(* Logix 5000 project; controller Modbus_TCP_Client_Example vendor 1 type 14 code 154 rev 32.15; software revision 32.05; part 6 of 10 *)

ADD_ON_INSTRUCTION AMP_Point_to_Point_IO_Servo   (* revision 1.0, vendor Applied Motion Products Inc. *)
// Applied Motion - Point to Point Move with IO AOI
// Help:
// The Point-to-Point Move with I/O AOI executes moves involving up to 2 Input conditions and a possible output state change. The move variant can be any of the following:
// - FS - Feed to Sensor
// - FD - Feed to Double Sensor
// - FM - Feed to Sensor with Mask Distance
// - FY - Feed to Sensor with Safety Distance
// - FO - Feed to Length and Set Output
// - SH - Seek Home
// All six(6) of the above variants need exactly one I/O point except for FD which requires a second I/O point to be specified in the parameters.
VAR_IN_OUT
   Input : DINT[20]; {required}   // Drive Input Assembly
        [16]   // Analog_Input1
        [4]   // Alarm_Code
        [0]   // Control_Word_Received
        [10]   // Position_Error
        [11]   // Actual_Velocity_RPS
        [12]   // Digital_Outputs
        [13]   // Digital_Inputs
        [14]   // Analog_Output1
        [15]   // Analog_Output2
        [17]   // Analog_Input2
        [18]   // Torque_Limit
        [19]   // Second_Encoder_Speed
        [1]   // OpCode1_Received
        [2]   // Control_Mode
        [3]   // Status_Code
        [5]   // Supply_Voltage
        [6]   // Applied_Torque
        [7]   // Drive_Temperature
        [8]   // Encoder_Position
        [9]   // Second_Encoder_Position
   Output : DINT[11]; {required}   // Drive Output Assembly
        [10]   // Reserved
        [4]   // Target Velocity
        [0]   // Control Word
        [3]   // Target Pos
        [1]   // OpCode 1
        [2]   // OpCode 2
        [5]   // Porifle Acceleration
        [6]   // Profile Deceleration
        [7]   // Target Torque
        [8]   // OpCode 3
        [9]   // OpCode 4
END_VAR
VAR_INPUT
   Start : BOOL; {required}   // Start the Move
   Command : INT := 'FS'; {required}   // Command variant: FS/FD/FY/FM/FO/SH
   IO1_Number : DINT; {required}   // Main Input/Output Number (0 = Encoder index, 1-8 = In/Out 1-8)
   IO1_Condition : SINT := 'R'; {required}   // Main Input/Output Condition/State H/L/R/F (High/Low/Rising Edge/Falling Edge)
   IO2_Number : DINT; {required}   // Second Input/Output Number (0 = Encoder index, 1-8 = In/Out 1-8)
   IO2_Condition : SINT; {required}   // Second Input/Output Condition/State H/L/R/F (High/Low/Rising Edge/Falling Edge)
   Distance : DINT; {required}   // Distance to Move (negative = reverse)
   Speed : REAL; {required}   // Velocity of Move (rev/sec)
   Acc : REAL; {required}   // Acceleration of Move (rev/s/s)
   Dec : REAL; {required}   // Deceleration (rev/s/s)
   Change_Distance : DINT; {required}   // Change Distance (steps, FY/FM/FO only)
   Change_Speed : REAL; {required}   // Velocity Change (rev/s) (FD only)
END_VAR
VAR_OUTPUT
   Sent : BOOL; {access Read Only, visible}   // Move has been sent to drive
   In_Progress : BOOL; {access Read Only, visible}   // Move in progress
   Done : BOOL; {access Read Only, visible}   // Move completed without errors - desired position reached
   Error : BOOL; {access Read Only, visible}   // Move failed to complete - drive not ready or faulted
   State : DINT := 10; {access Read Only}   // Internal state of progress
END_VAR
VAR
   Loc_StatusCode : AMP_Status_Word_Servo; {access None}
   Loc_Start_ONS : BOOL; {access None}
   Loc_Input_Assembly : AMP_Input_Assembly_Servo_v2; {access None}
   Loc_Command_Timeout : TIMER := (PRE := 2000); {access None}   // Timer to output fault if command is not Done
   Loc_ChangeSpeed_Required : BOOL; {access None}
   Loc_ChangeDistance_Required : BOOL; {access None}
   Loc_IO2_Number_Encoded : DINT; {access None}
   Loc_IO2_Condition_Encoded : DINT; {access None}
   Loc_IO1_Condition_Encoded : DINT; {access None}
   Loc_IO1_Number_Encoded : DINT; {access None}
END_VAR

ROUTINE Logic   (* ladder *)
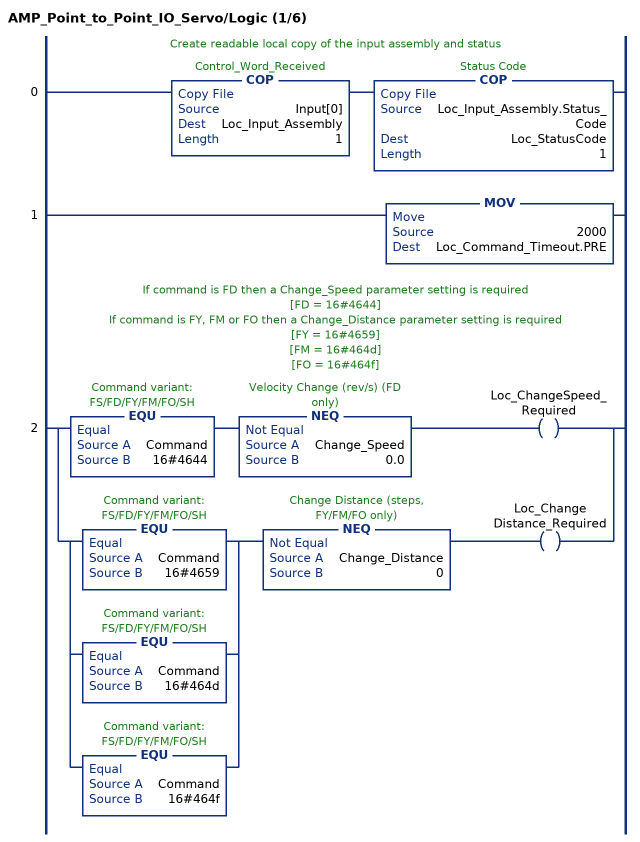
   // Create readable local copy of the input assembly and status
   0: COP(Input[0],Loc_Input_Assembly,1)COP(Loc_Input_Assembly.Status_Code,Loc_StatusCode,1);
   1: MOV(2000,Loc_Command_Timeout.PRE);
   // If command is FD then a Change_Speed parameter setting is required
   // [FD = 16#4644]
   // If command is FY, FM or FO then a Change_Distance parameter setting is required
   // [FY = 16#4659]
   // [FM = 16#464d]
   // [FO = 16#464f]
   2: [EQU(Command,16#4644) NEQ(Change_Speed,0.0) OTE(Loc_ChangeSpeed_Required) ,[EQU(Command,16#4659) ,EQU(Command,16#464d) ,EQU(Command,16#464f) ] NEQ(Change_Distance,0) OTE(Loc_ChangeDistance_Required) ];
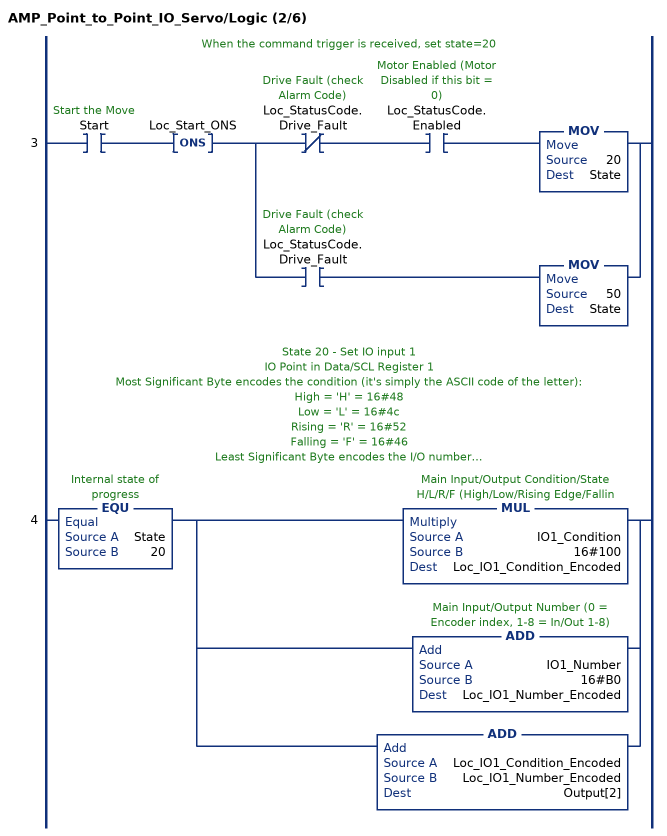
   // When the command trigger is received, set state=20
   3: XIC(Start)ONS(Loc_Start_ONS)[XIO(Loc_StatusCode.Drive_Fault) XIC(Loc_StatusCode.Enabled) MOV(20,State) ,XIC(Loc_StatusCode.Drive_Fault) MOV(50,State) ];
   // State 20 - Set IO input 1
   // IO Point in Data/SCL Register 1
   // Most Significant Byte encodes the condition (it's simply the ASCII code of the letter):
   // High = 'H' = 16#48
   // Low = 'L' = 16#4c
   // Rising = 'R' = 16#52
   // Falling = 'F' = 16#46
   // Least Significant Byte encodes the I/O number:
   // 0xB0-0xBC for connector  (IN/OUT1) depending on provided I/O number 0-12 (0=encoder)
   4: EQU(State,20)[MUL(IO1_Condition,16#100,Loc_IO1_Condition_Encoded) ,ADD(IO1_Number,16#B0,Loc_IO1_Number_Encoded) ,ADD(Loc_IO1_Condition_Encoded,Loc_IO1_Number_Encoded,Output[2]) ];
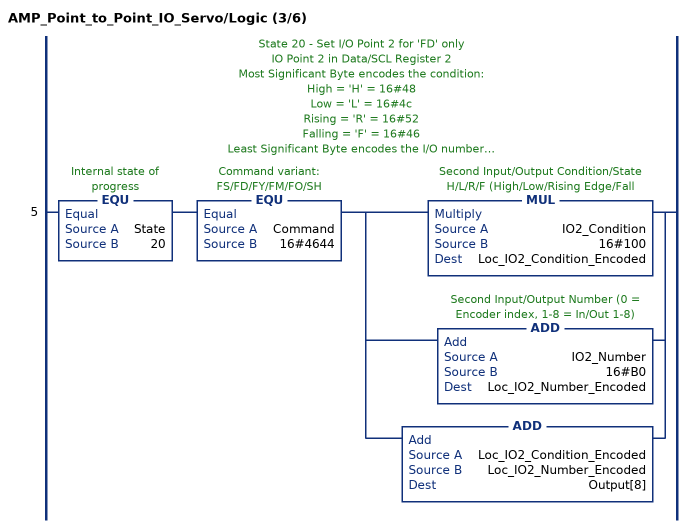
   // State 20 - Set I/O Point 2 for 'FD' only
   // IO Point 2 in Data/SCL Register 2
   // Most Significant Byte encodes the condition:
   // High = 'H' = 16#48
   // Low = 'L' = 16#4c
   // Rising = 'R' = 16#52
   // Falling = 'F' = 16#46
   // Least Significant Byte encodes the I/O number:
   // 0xB0-0xBC for connector  (IN/OUT1) depending on provided I/O number 0-12 (0=encoder)
   5: EQU(State,20)EQU(Command,16#4644)[MUL(IO2_Condition,16#100,Loc_IO2_Condition_Encoded) ,ADD(IO2_Number,16#B0,Loc_IO2_Number_Encoded) ,ADD(Loc_IO2_Condition_Encoded,Loc_IO2_Number_Encoded,Output[8]) ];
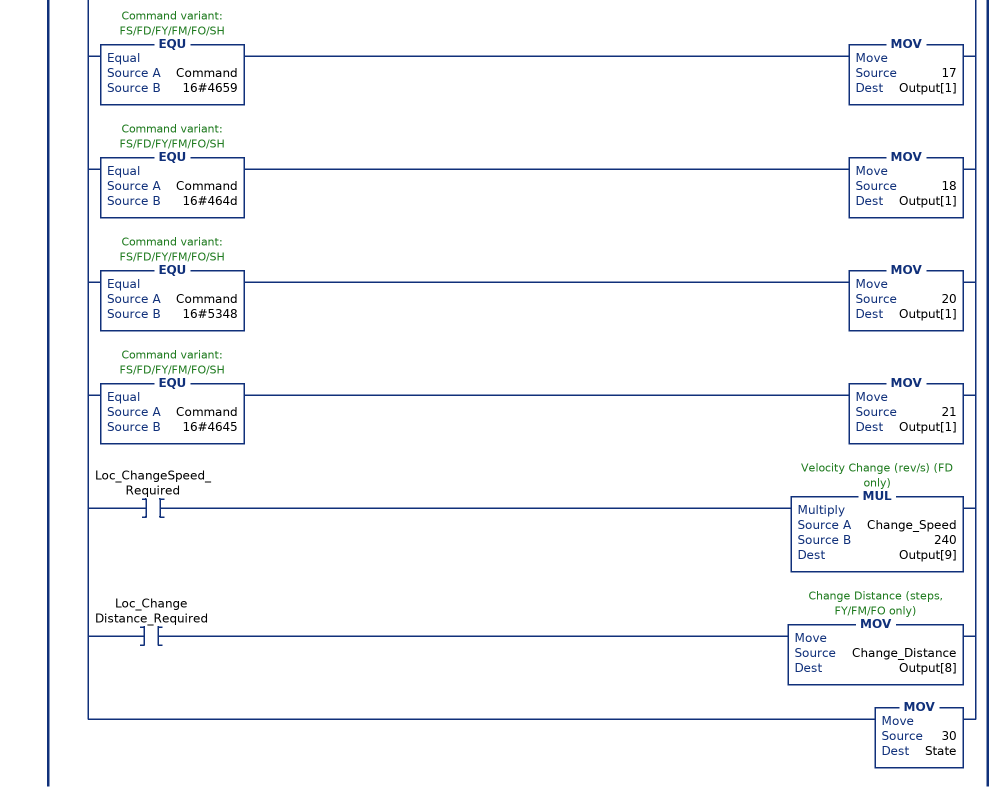
   // State 20 -
   // Distance in motor steps, no conversion required
   // Speed in rev/s, converted to 0.25 rev/min
   // Acceleration in rev/s/s, converted to 10 rev/min/s
   // Deceleration in rev/s/s, converted to 10 rev/min/s
   // FS (Feed to Sensor): ASCII = 16#4653, Cmd = 12,
   // FO (Feed to Length and Set Output): ASCII = 16#464f, Cmd = 13,
   // FD (Feed to Double Sensor): ASCII = 16#4644, Cmd = 16,
   // FY (Feed to Sensor with Safety Distance): ASCII = 16#4659, Cmd = 17,
   // FM (Feed to Sensor with Mask Distance): ASCII = 16#464d, Cmd = 18,
   // SH (Seek Home): ASCII = 16#5348, Cmd = 20
   6: EQU(State,20)EQU(Loc_Input_Assembly.Control_Mode,21)ADD(Loc_Input_Assembly.Control_Word_Received,1,Output[0])[MOV(Distance,Output[3]) ,MUL(Speed,240,Output[4]) ,MUL(Acc,6,Output[5]) ,MUL(Dec,6,Output[6]) ][[EQU(Command,16#4653) MOV(12,Output[1]) ,EQU(Command,16#464f) MOV(13,Output[1]) ,EQU(Command,16#4644) MOV(16,Output[1]) ,EQU(Command,16#4659) MOV(17,Output[1]) ,EQU(Command,16#464d) MOV(18,Output[1]) ,EQU(Command,16#5348) MOV(20,Output[1]) ,EQU(Command,16#4645) MOV(21,Output[1]) ] ,XIC(Loc_ChangeSpeed_Required) MUL(Change_Speed,240,Output[9]) ,XIC(Loc_ChangeDistance_Required) MOV(Change_Distance,Output[8]) ,MOV(30,State) ];
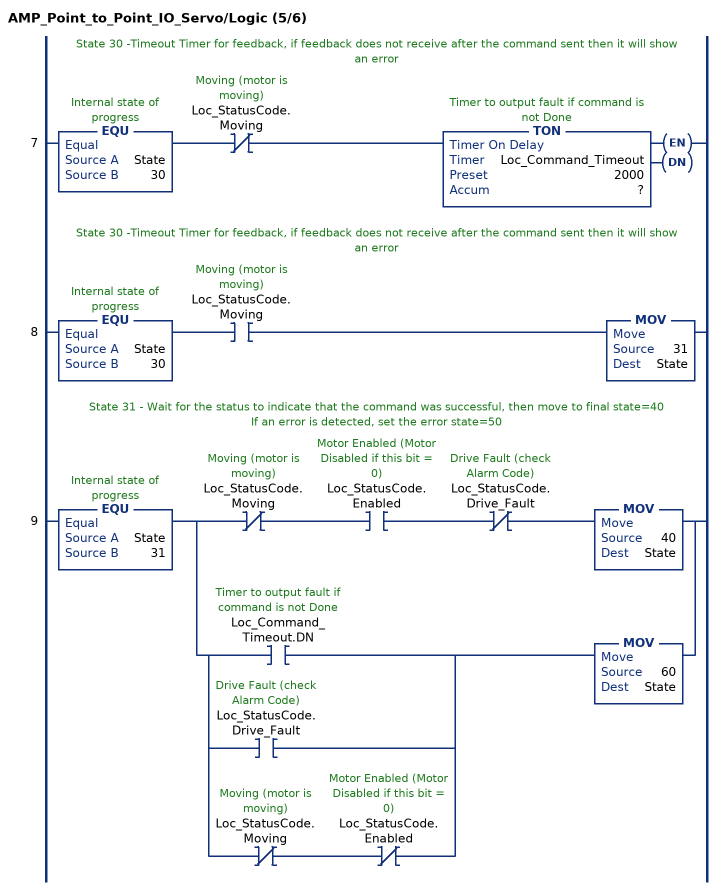
   // State 30 -Timeout Timer for feedback, if feedback does not receive after the command sent then it will show an error
   7: EQU(State,30)XIO(Loc_StatusCode.Moving)TON(Loc_Command_Timeout,?,?);
   // State 30 -Timeout Timer for feedback, if feedback does not receive after the command sent then it will show an error
   8: EQU(State,30)XIC(Loc_StatusCode.Moving)MOV(31,State);
   // State 31 - Wait for the status to indicate that the command was successful, then move to final state=40
   // If an error is detected, set the error state=50
   9: EQU(State,31)[XIO(Loc_StatusCode.Moving) XIC(Loc_StatusCode.Enabled) XIO(Loc_StatusCode.Drive_Fault) MOV(40,State) ,[XIC(Loc_Command_Timeout.DN) ,XIC(Loc_StatusCode.Drive_Fault) ,XIO(Loc_StatusCode.Moving) XIO(Loc_StatusCode.Enabled) ] MOV(60,State) ];
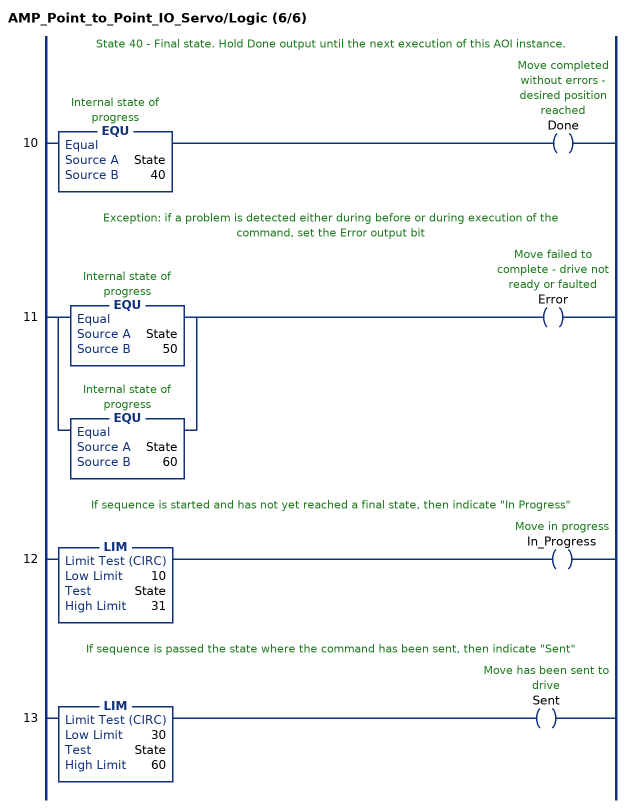
   // State 40 - Final state. Hold Done output until the next execution of this AOI instance.
   10: EQU(State,40)OTE(Done);
   // Exception: if a problem is detected either during before or during execution of the command, set the Error output bit
   11: [EQU(State,50) ,EQU(State,60) ]OTE(Error);
   // If sequence is started and has not yet reached a final state, then indicate "In Progress"
   12: LIM(10,State,31)OTE(In_Progress);
   // If sequence is passed the state where the command has been sent, then indicate "Sent"
   13: LIM(30,State,60)OTE(Sent);
END_ROUTINE
END_ADD_ON_INSTRUCTION

ADD_ON_INSTRUCTION AMP_Q_Segment_Execute   (* revision 1.0 *)
// Applied Motion - Q Segment Execute AOI
// Help:
// The SCL Command Execute AOI executes selected SCL commands (as listed under “Available SCL Commands” in the Host Command Reference).
VAR_IN_OUT
   Input : DINT[14]; {required}   // Drive Input Assembly
   Output : DINT[16]; {required}   // Drive Output Assembly
        [0]   // Command Word
        [10]   // Data/Register 1
        [11]   // Data/Register 2
        [1]   // Jog Speed (0.25 rev/min)
        [2]   // Jog Acceleration (10 rev/s/s)
        [3]   // Jog Deceleration (10 rev/s/s)
        [4]   // Point-to-Point Velocity (0.25 rev/min)
        [5]   // Point-to-Point Acceleration (10 rev/s/s)
        [6]   // Point-to-Point Deceleration (10 rev/s/s)
        [7]   // Point-to-Point Distance (Motor steps)
        [9]   // (2x ASCII Letters in 16 lower word)
END_VAR
VAR_INPUT
   RPI : DINT := 100; {visible}   // Drive Connection Request Packet Interval (milliseconds)
   LoadAndExec : BOOL; {required}   // Load and Execute the specified Q segment (edge triggered)
   Q_Segment : DINT; {required}   // Q Segment to Load and Execute
END_VAR
VAR_OUTPUT
   Sent : BOOL; {access Read Only, visible}   // Command has been sent to drive
   In_Progress : BOOL; {access Read Only, visible}   // In progress = sending command
   Done : BOOL; {access Read Only, visible}   // Command sent
   Error : BOOL; {access Read Only, visible}   // Command failed to be sent
   State : DINT := 10; {access Read Only}   // Internal state of progress
END_VAR
VAR
   Loc_StatusCode : AMP_Status_Word;
   Loc_CommandOff_Timer : TIMER;   // Timer to make sure command value was 0 before sending a new command
   Loc_CommandOn_Timer : TIMER;   // Timer to make sure command value is set long enough to be sent to drive
   Loc_Input_Assembly : AMP_Input_Assembly_v2; {access None}
   Loc_Start_ONS : BOOL; {access None}
END_VAR

ROUTINE Logic   (* ladder *)
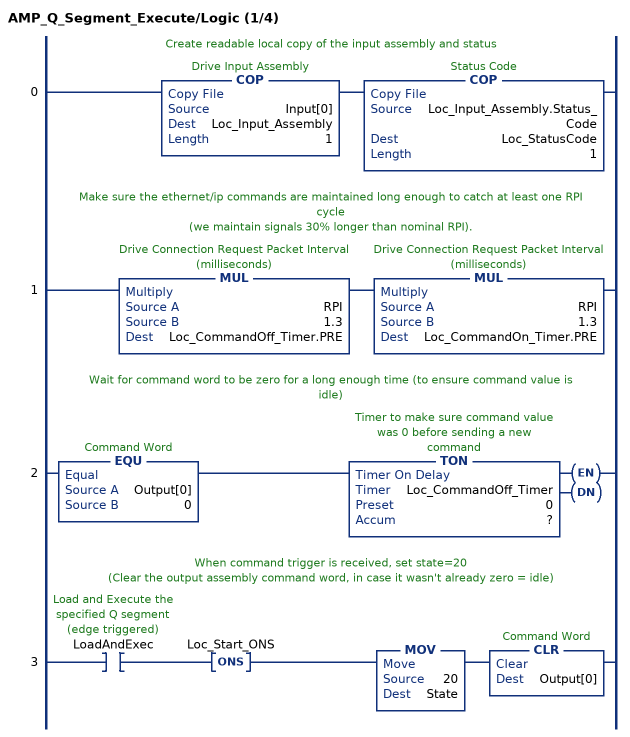
   // Create readable local copy of the input assembly and status
   0: COP(Input[0],Loc_Input_Assembly,1)COP(Loc_Input_Assembly.Status_Code,Loc_StatusCode,1);
   // Make sure the ethernet/ip commands are maintained long enough to catch at least one RPI cycle
   // (we maintain signals 30% longer than nominal RPI).
   1: MUL(RPI,1.3,Loc_CommandOff_Timer.PRE)MUL(RPI,1.3,Loc_CommandOn_Timer.PRE);
   // Wait for command word to be zero for a long enough time (to ensure command value is idle)
   2: EQU(Output[0],0)TON(Loc_CommandOff_Timer,?,?);
   // When command trigger is received, set state=20
   // (Clear the output assembly command word, in case it wasn't already zero = idle)
   3: XIC(LoadAndExec)ONS(Loc_Start_ONS)MOV(20,State)CLR(Output[0]);
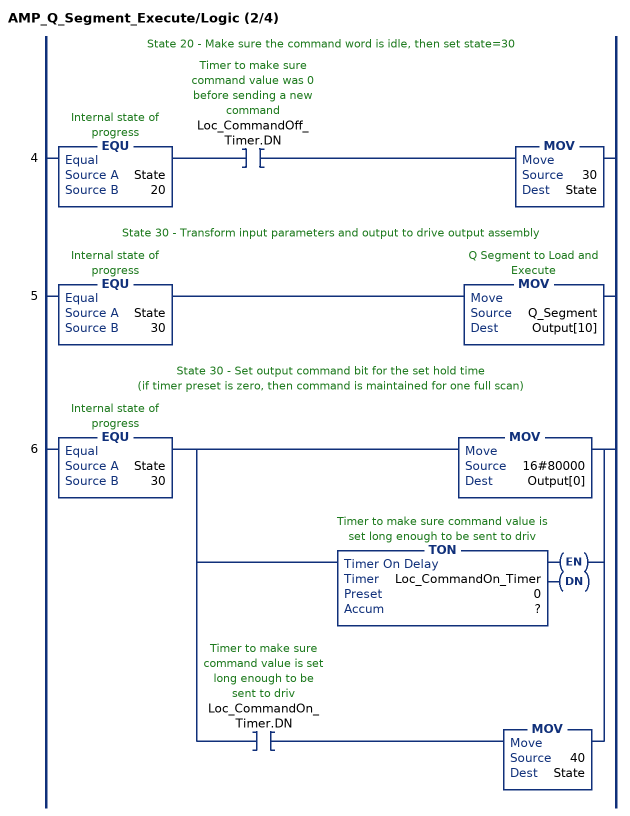
   // State 20 - Make sure the command word is idle, then set state=30
   4: EQU(State,20)XIC(Loc_CommandOff_Timer.DN)MOV(30,State);
   // State 30 - Transform input parameters and output to drive output assembly
   5: EQU(State,30)MOV(Q_Segment,Output[10]);
   // State 30 - Set output command bit for the set hold time
   // (if timer preset is zero, then command is maintained for one full scan)
   6: EQU(State,30)[MOV(16#80000,Output[0]) ,TON(Loc_CommandOn_Timer,?,?) ,XIC(Loc_CommandOn_Timer.DN) MOV(40,State) ];
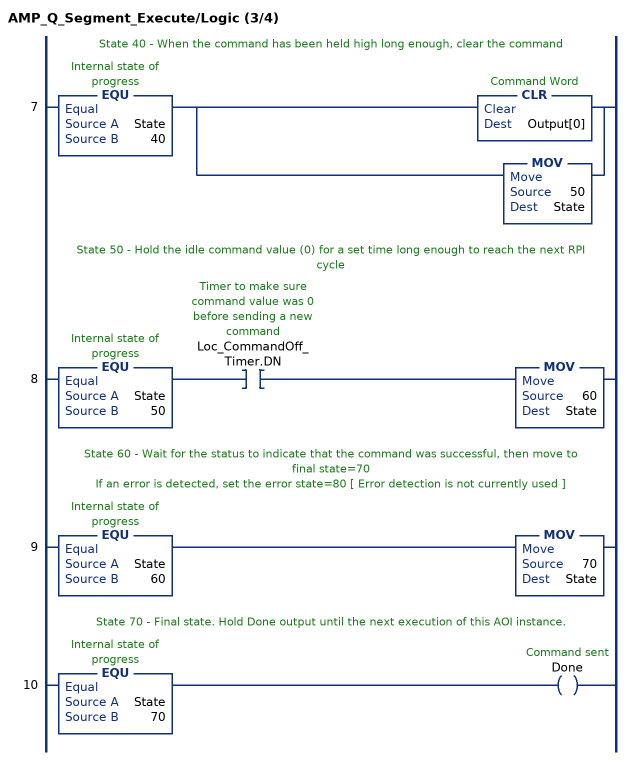
   // State 40 - When the command has been held high long enough, clear the command
   7: EQU(State,40)[CLR(Output[0]) ,MOV(50,State) ];
   // State 50 - Hold the idle command value (0) for a set time long enough to reach the next RPI cycle
   8: EQU(State,50)XIC(Loc_CommandOff_Timer.DN)MOV(60,State);
   // State 60 - Wait for the status to indicate that the command was successful, then move to final state=70
   // If an error is detected, set the error state=80 [ Error detection is not currently used ]
   9: EQU(State,60)MOV(70,State);
   // State 70 - Final state. Hold Done output until the next execution of this AOI instance.
   10: EQU(State,70)OTE(Done);
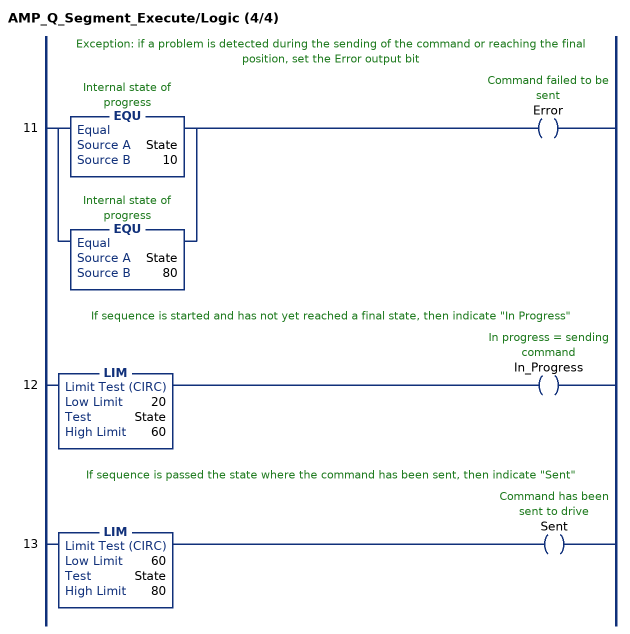
   // Exception: if a problem is detected during the sending of the command or reaching the final position, set the Error output bit
   11: [EQU(State,10) ,EQU(State,80) ]OTE(Error);
   // If sequence is started and has not yet reached a final state, then indicate "In Progress"
   12: LIM(20,State,60)OTE(In_Progress);
   // If sequence is passed the state where the command has been sent, then indicate "Sent"
   13: LIM(60,State,80)OTE(Sent);
END_ROUTINE
END_ADD_ON_INSTRUCTION

ADD_ON_INSTRUCTION AMP_Q_Segment_Execute_Servo   (* revision 1.0, vendor Applied Motion Products Inc. *)
// Applied Motion - Q Segment Execute AOI
// Help:
// This AOI Execute Q program Segment. Q program are written inside the drive using Applied Motion software.
VAR_IN_OUT
   Input : DINT[20]; {required}   // Drive Input Assembly
        [4]   // Alarm_Code
        [16]   // Analog_Input1
        [0]   // Control_Word_Received
        [10]   // Position_Error
        [11]   // Actual_Velocity_RPS
        [12]   // Digital_Outputs
        [13]   // Digital_Inputs
        [14]   // Analog_Output1
        [15]   // Analog_Output2
        [17]   // Analog_Input2
        [18]   // Torque_Limit
        [19]   // Second_Encoder_Speed
        [1]   // OpCode1_Received
        [2]   // Control_Mode
        [3]   // Status_Code
        [5]   // Supply_Voltage
        [6]   // Applied_Torque
        [7]   // Drive_Temperature
        [8]   // Encoder_Position
        [9]   // Second_Encoder_Position
   Output : DINT[11]; {required}   // Drive Output Assembly
        [10]   // Reserved
        [4]   // Target Velocity
        [0]   // Control Word
        [3]   // Target Pos
        [1]   // OpCode 1
        [2]   // OpCode 2
        [5]   // Porifle Acceleration
        [6]   // Profile Deceleration
        [7]   // Target Torque
        [8]   // OpCode 3
        [9]   // OpCode 4
END_VAR
VAR_INPUT
   LoadAndExec : BOOL; {required}   // Load and Execute the specified Q segment (edge triggered)
   Q_Segment : DINT; {required}   // Q Segment to Load and Execute
END_VAR
VAR_OUTPUT
   Sent : BOOL; {access Read Only, visible}   // Command has been sent to drive
   In_Progress : BOOL; {access Read Only, visible}   // In progress = sending command
   Done : BOOL; {access Read Only, visible}   // Command sent
   Error : BOOL; {access Read Only, visible}   // Command failed to be sent
   State : DINT := 10; {access Read Only}   // Internal state of progress
END_VAR
VAR
   Loc_StatusCode : AMP_Status_Word_Servo; {access None}
   Loc_Q_Exe_ONS : BOOL;
   Loc_Input_Assembly : AMP_Input_Assembly_Servo_v2; {access None}
END_VAR

ROUTINE Logic   (* ladder *)
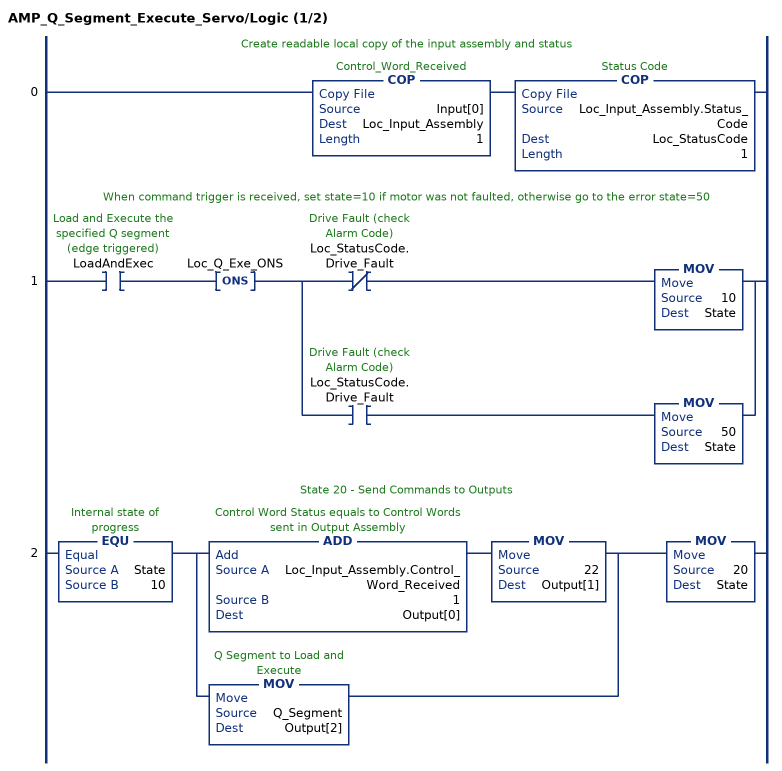
   // Create readable local copy of the input assembly and status
   0: COP(Input[0],Loc_Input_Assembly,1)COP(Loc_Input_Assembly.Status_Code,Loc_StatusCode,1);
   // When command trigger is received, set state=10 if motor was not faulted, otherwise go to the error state=50
   1: XIC(LoadAndExec)ONS(Loc_Q_Exe_ONS)[XIO(Loc_StatusCode.Drive_Fault) MOV(10,State) ,XIC(Loc_StatusCode.Drive_Fault) MOV(50,State) ];
   // State 20 - Send Commands to Outputs
   2: EQU(State,10)[ADD(Loc_Input_Assembly.Control_Word_Received,1,Output[0]) MOV(22,Output[1]) ,MOV(Q_Segment,Output[2]) ]MOV(20,State);
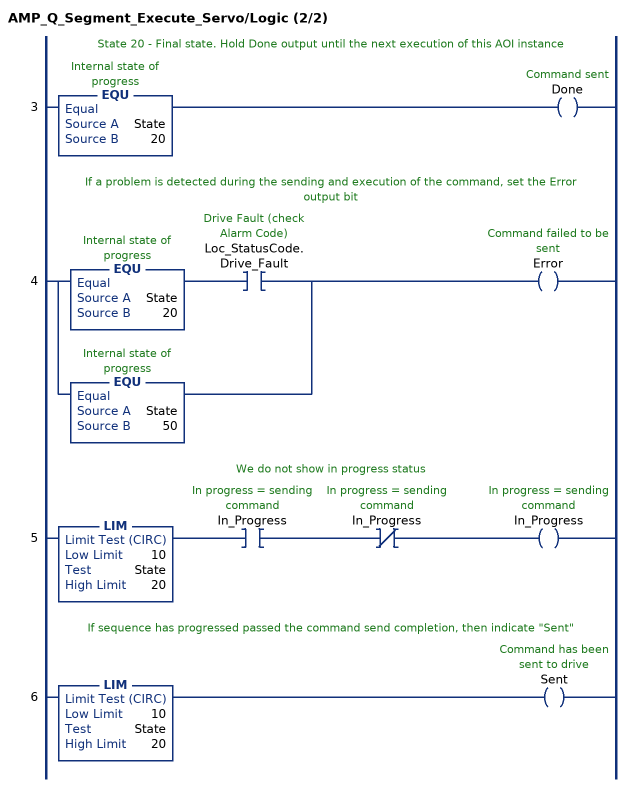
   // State 20 - Final state. Hold Done output until the next execution of this AOI instance
   3: EQU(State,20)OTE(Done);
   // If a problem is detected during the sending and execution of the command, set the Error output bit
   4: [EQU(State,20) XIC(Loc_StatusCode.Drive_Fault) ,EQU(State,50) ]OTE(Error);
   // We do not show in progress status
   5: LIM(10,State,20)XIC(In_Progress)XIO(In_Progress)OTE(In_Progress);
   // If sequence has progressed passed the command send completion, then indicate "Sent"
   6: LIM(10,State,20)OTE(Sent);
END_ROUTINE
END_ADD_ON_INSTRUCTION

ADD_ON_INSTRUCTION AMP_Relative_Move   (* revision 1.0 *)
// Applied Motion - Relative Move AOI
// Help:
// The Relative Move AOI is used to move an axis by a specified distance (positive or negative) relative to its currently commanded position.
VAR_IN_OUT
   Input : DINT[14]; {required}   // Drive Input Assembly
   Output : DINT[16]; {required}   // Drive Output Assembly
        [0]   // Command Word
        [10]   // Data/Register 1
        [11]   // Data/Register 2
        [1]   // Jog Speed (0.25 rev/min)
        [2]   // Jog Acceleration (10 rev/s/s)
        [3]   // Jog Deceleration (10 rev/s/s)
        [4]   // Point-to-Point Velocity (0.25 rev/min)
        [5]   // Point-to-Point Acceleration (10 rev/min/s)
        [6]   // Point-to-Point Deceleration (10 rev/min/s)
        [7]   // Point-to-Point Distance (Motor steps)
        [9]   // (2x ASCII Letters in 16 lower word)
END_VAR
VAR_INPUT
   RPI : DINT := 100; {visible}   // Drive Connection Request Packet Interval (milliseconds)
   Start : BOOL; {required}   // Start the Relative Move
   Distance : DINT; {required}   // Relative Distance to Move (steps, negative = reverse)
   Speed : REAL; {required}   // Velocity of Move (rev/min)
   Acc : REAL; {required}   // Acceleration of Move (rev/s/s)
   Dec : REAL; {required}   // Deceleration (rev/s/s)
END_VAR
VAR_OUTPUT
   Sent : BOOL; {access Read Only, visible}   // Move has been sent to drive
   In_Progress : BOOL; {access Read Only, visible}   // Move in progress
   Done : BOOL; {access Read Only, visible}   // Move completed without errors - desired position reached
   Error : BOOL; {access Read Only, visible}   // Move failed to complete - drive not ready or faulted
   State : DINT := 10; {access Read Only}   // Internal state of progress
END_VAR
VAR
   Loc_StatusCode : AMP_Status_Word;
   Loc_CommandOff_Timer : TIMER;   // Timer to make sure command value was 0 before sending a new command
   Loc_CommandOn_Timer : TIMER;   // Timer to make sure command value is set long enough to be sent to drive
   Loc_Input_Assembly : AMP_Input_Assembly_v2; {access None}
   Loc_Start_ONS : BOOL; {access None}
   Loc_AlarmCode : AMP_Alarm_Word; {access None}
END_VAR

ROUTINE Logic   (* ladder *)
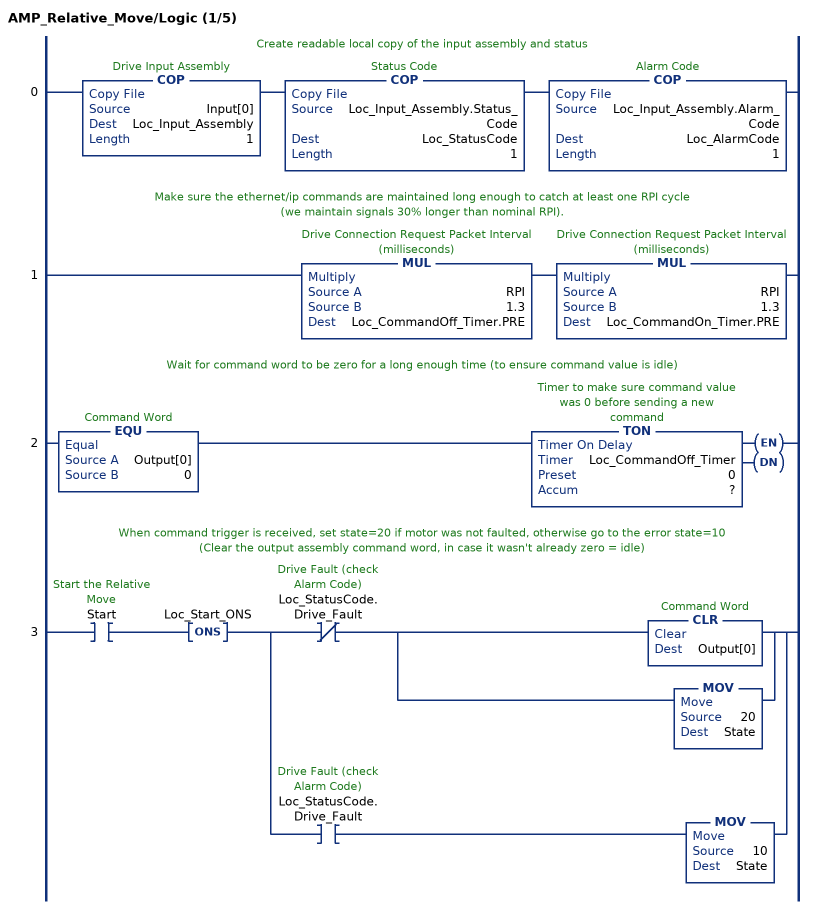
   // Create readable local copy of the input assembly and status
   0: COP(Input[0],Loc_Input_Assembly,1)COP(Loc_Input_Assembly.Status_Code,Loc_StatusCode,1)COP(Loc_Input_Assembly.Alarm_Code,Loc_AlarmCode,1);
   // Make sure the ethernet/ip commands are maintained long enough to catch at least one RPI cycle
   // (we maintain signals 30% longer than nominal RPI).
   1: MUL(RPI,1.3,Loc_CommandOff_Timer.PRE)MUL(RPI,1.3,Loc_CommandOn_Timer.PRE);
   // Wait for command word to be zero for a long enough time (to ensure command value is idle)
   2: EQU(Output[0],0)TON(Loc_CommandOff_Timer,?,?);
   // When command trigger is received, set state=20 if motor was not faulted, otherwise go to the error state=10
   // (Clear the output assembly command word, in case it wasn't already zero = idle)
   3: XIC(Start)ONS(Loc_Start_ONS)[XIO(Loc_StatusCode.Drive_Fault) [CLR(Output[0]) ,MOV(20,State) ] ,XIC(Loc_StatusCode.Drive_Fault) MOV(10,State) ];
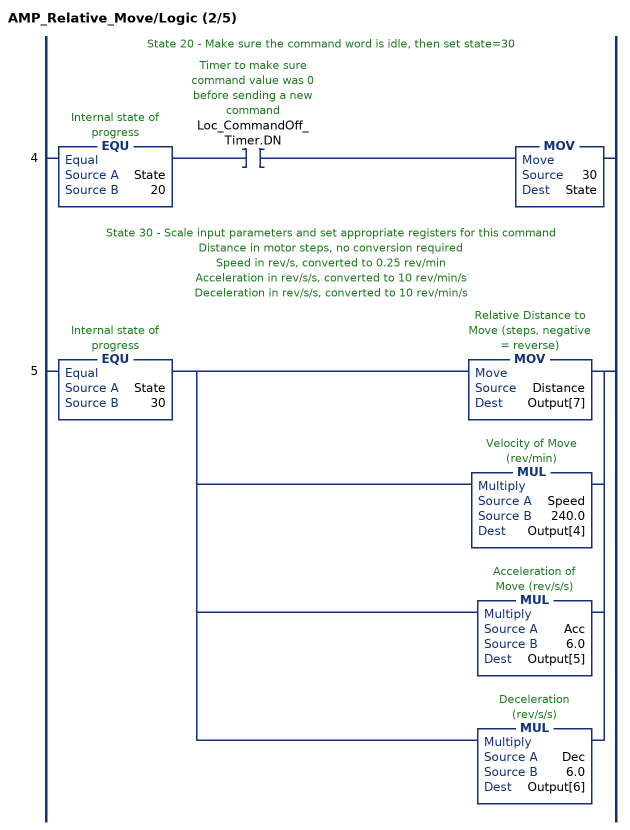
   // State 20 - Make sure the command word is idle, then set state=30
   4: EQU(State,20)XIC(Loc_CommandOff_Timer.DN)MOV(30,State);
   // State 30 - Scale input parameters and set appropriate registers for this command
   // Distance in motor steps, no conversion required
   // Speed in rev/s, converted to 0.25 rev/min
   // Acceleration in rev/s/s, converted to 10 rev/min/s
   // Deceleration in rev/s/s, converted to 10 rev/min/s
   5: EQU(State,30)[MOV(Distance,Output[7]) ,MUL(Speed,240.0,Output[4]) ,MUL(Acc,6.0,Output[5]) ,MUL(Dec,6.0,Output[6]) ];
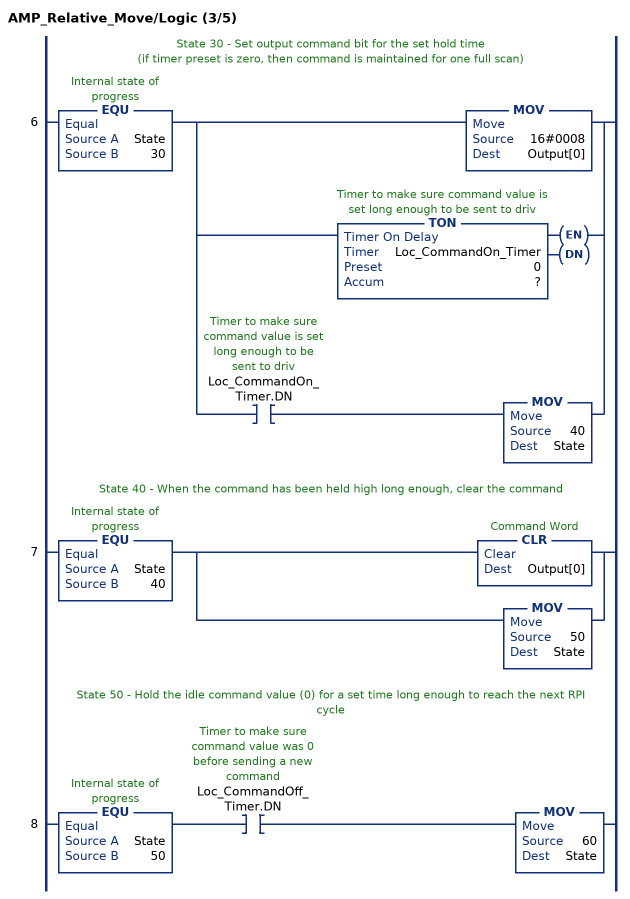
   // State 30 - Set output command bit for the set hold time
   // (if timer preset is zero, then command is maintained for one full scan)
   6: EQU(State,30)[MOV(16#0008,Output[0]) ,TON(Loc_CommandOn_Timer,?,?) ,XIC(Loc_CommandOn_Timer.DN) MOV(40,State) ];
   // State 40 - When the command has been held high long enough, clear the command
   7: EQU(State,40)[CLR(Output[0]) ,MOV(50,State) ];
   // State 50 - Hold the idle command value (0) for a set time long enough to reach the next RPI cycle
   8: EQU(State,50)XIC(Loc_CommandOff_Timer.DN)MOV(60,State);
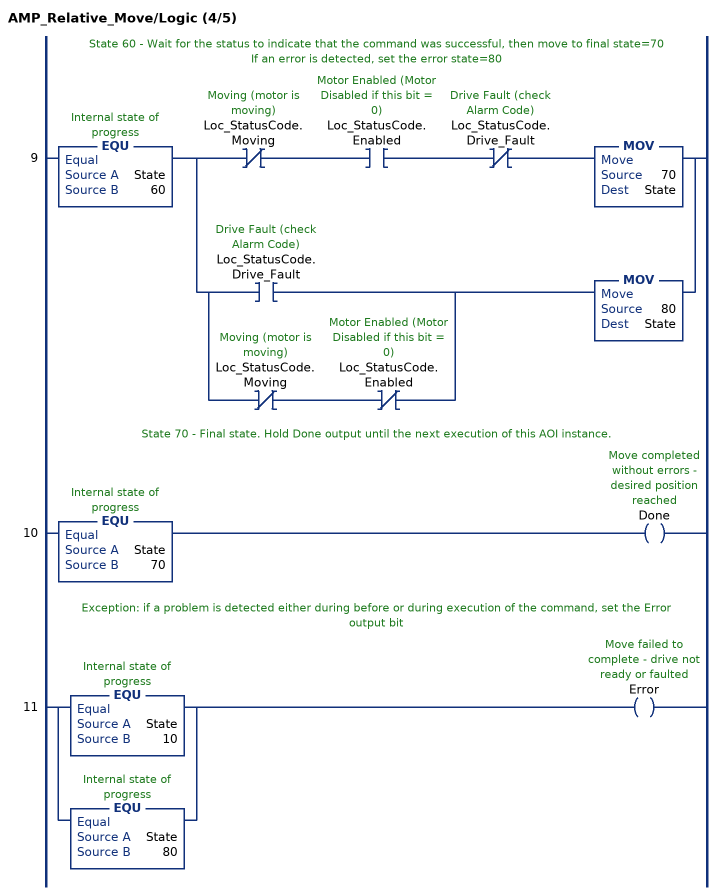
   // State 60 - Wait for the status to indicate that the command was successful, then move to final state=70
   // If an error is detected, set the error state=80
   9: EQU(State,60)[XIO(Loc_StatusCode.Moving) XIC(Loc_StatusCode.Enabled) XIO(Loc_StatusCode.Drive_Fault) MOV(70,State) ,[XIC(Loc_StatusCode.Drive_Fault) ,XIO(Loc_StatusCode.Moving) XIO(Loc_StatusCode.Enabled) ] MOV(80,State) ];
   // State 70 - Final state. Hold Done output until the next execution of this AOI instance.
   10: EQU(State,70)OTE(Done);
   // Exception: if a problem is detected either during before or during execution of the command, set the Error output bit
   11: [EQU(State,10) ,EQU(State,80) ]OTE(Error);
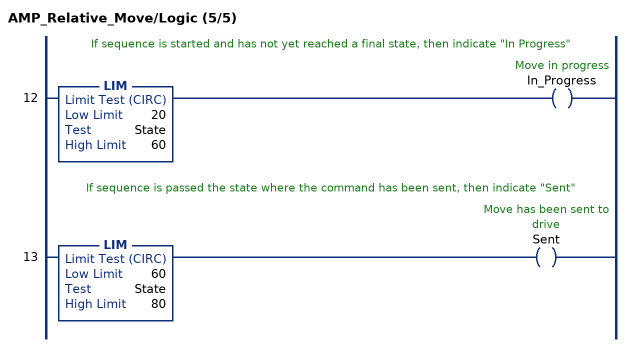
   // If sequence is started and has not yet reached a final state, then indicate "In Progress"
   12: LIM(20,State,60)OTE(In_Progress);
   // If sequence is passed the state where the command has been sent, then indicate "Sent"
   13: LIM(60,State,80)OTE(Sent);
END_ROUTINE
END_ADD_ON_INSTRUCTION

ADD_ON_INSTRUCTION AMP_Relative_Move_Servo   (* revision 1.0, vendor Applied Motion Products Inc. *)
// Applied Motion - Motor Relative Move - AOI
// Help:
// The Relative Move AOI is used to move an axis by a specified distance (positive or negative) relative to its currently commanded position(FL).
VAR_IN_OUT
   Input : DINT[20]; {required}   // Drive Input Assembly
        [16]   // Analog_Input1
        [4]   // Alarm_Code
        [0]   // Control_Word_Received
        [10]   // Position_Error
        [11]   // Actual_Velocity_RPS
        [12]   // Digital_Outputs
        [13]   // Digital_Inputs
        [14]   // Analog_Output1
        [15]   // Analog_Output2
        [17]   // Analog_Input2
        [18]   // Torque_Limit
        [19]   // Second_Encoder_Speed
        [1]   // OpCode1_Received
        [2]   // Control_Mode
        [3]   // Status_Code
        [5]   // Supply_Voltage
        [6]   // Applied_Torque
        [7]   // Drive_Temperature
        [8]   // Encoder_Position
        [9]   // Second_Encoder_Position
   Output : DINT[11]; {required}   // Drive Output Assembly
        [10]   // Reserved
        [4]   // Target Velocity
        [0]   // Control Word
        [3]   // Target Pos
        [1]   // OpCode 1
        [2]   // OpCode 2
        [5]   // Porifle Acceleration
        [6]   // Profile Deceleration
        [7]   // Target Torque
        [8]   // OpCode 3
        [9]   // OpCode 4
END_VAR
VAR_INPUT
   Start : BOOL; {required}   // Start the Relative Move
   Distance : DINT; {required}   // Relative Distance to Move (negative = reverse)
   Speed_rps : REAL; {required}   // Velocity of Move (rev/sec)
   Acc : REAL; {required}   // Acceleration of Move (rev/s/s)
   Dec : REAL; {required}   // Deceleration of Move (rev/s/s)
END_VAR
VAR_OUTPUT
   Sent : BOOL; {access Read Only, visible}   // Move has been sent to drive
   In_Progress : BOOL; {access Read Only, visible}   // Move in progress
   Done : BOOL; {access Read Only, visible}   // Move completed without errors - desired position reached
   Error : BOOL; {access Read Only, visible}   // Move failed to complete - drive not ready or faulted
   State : DINT := 10; {access Read Only}   // Internal state of progress
END_VAR
VAR
   Loc_StatusCode : AMP_Status_Word_Servo; {access None}
   Loc_Rel_ONS : BOOL;
   Loc_Input_Assembly : AMP_Input_Assembly_Servo_v2; {access None}
   Loc_Command_Timeout : TIMER := (PRE := 2000); {access None}   // Timer to output fault if command is not Done
END_VAR

ROUTINE Logic   (* ladder *)
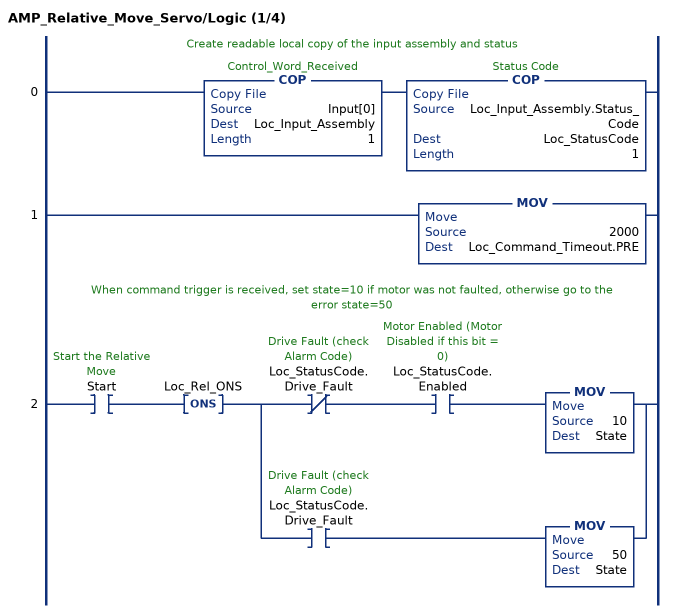
   // Create readable local copy of the input assembly and status
   0: COP(Input[0],Loc_Input_Assembly,1)COP(Loc_Input_Assembly.Status_Code,Loc_StatusCode,1);
   1: MOV(2000,Loc_Command_Timeout.PRE);
   // When command trigger is received, set state=10 if motor was not faulted, otherwise go to the error state=50
   2: XIC(Start)ONS(Loc_Rel_ONS)[XIO(Loc_StatusCode.Drive_Fault) XIC(Loc_StatusCode.Enabled) MOV(10,State) ,XIC(Loc_StatusCode.Drive_Fault) MOV(50,State) ];
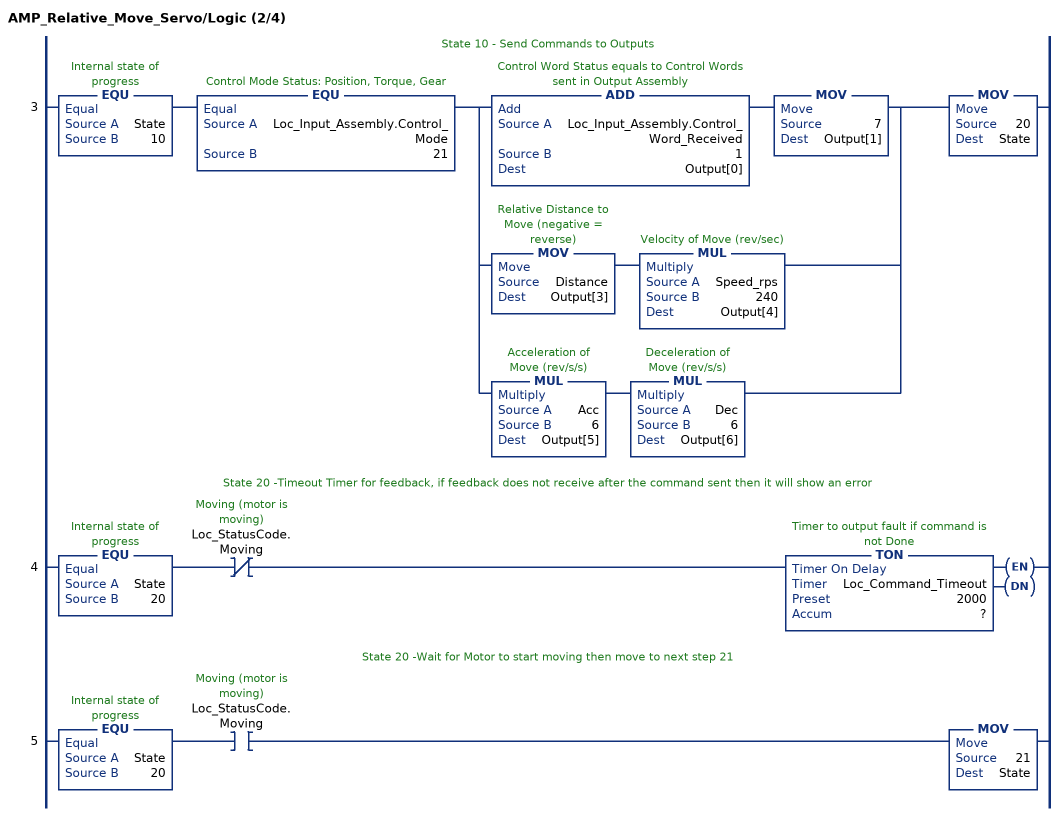
   // State 10 - Send Commands to Outputs
   3: EQU(State,10)EQU(Loc_Input_Assembly.Control_Mode,21)[ADD(Loc_Input_Assembly.Control_Word_Received,1,Output[0]) MOV(7,Output[1]) ,MOV(Distance,Output[3]) MUL(Speed_rps,240,Output[4]) ,MUL(Acc,6,Output[5]) MUL(Dec,6,Output[6]) ]MOV(20,State);
   // State 20 -Timeout Timer for feedback, if feedback does not receive after the command sent then it will show an error
   4: EQU(State,20)XIO(Loc_StatusCode.Moving)TON(Loc_Command_Timeout,?,?);
   // State 20 -Wait for Motor to start moving then move to next step 21
   5: EQU(State,20)XIC(Loc_StatusCode.Moving)MOV(21,State);
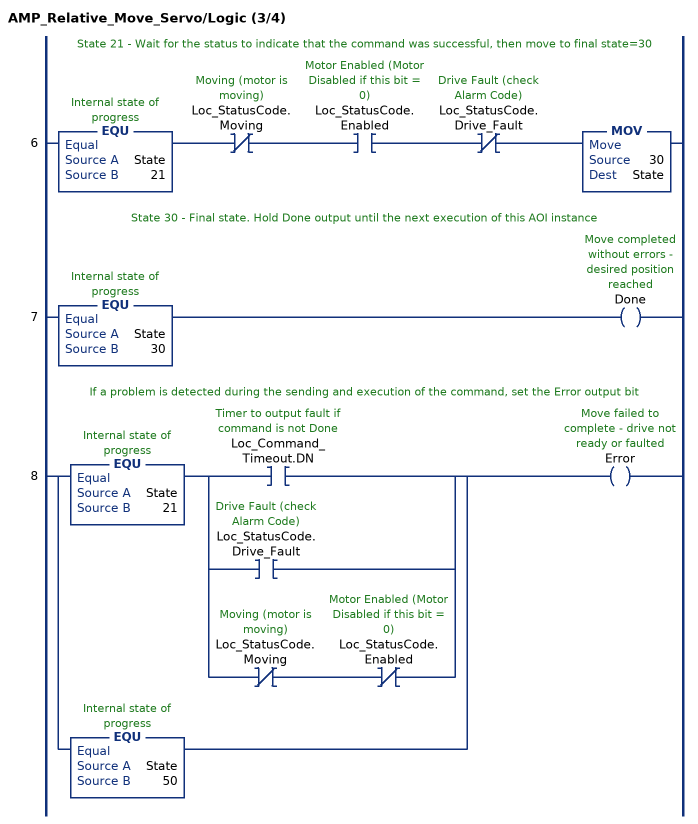
   // State 21 - Wait for the status to indicate that the command was successful, then move to final state=30
   6: EQU(State,21)XIO(Loc_StatusCode.Moving)XIC(Loc_StatusCode.Enabled)XIO(Loc_StatusCode.Drive_Fault)MOV(30,State);
   // State 30 - Final state. Hold Done output until the next execution of this AOI instance
   7: EQU(State,30)OTE(Done);
   // If a problem is detected during the sending and execution of the command, set the Error output bit
   8: [EQU(State,21) [XIC(Loc_Command_Timeout.DN) ,XIC(Loc_StatusCode.Drive_Fault) ,XIO(Loc_StatusCode.Moving) XIO(Loc_StatusCode.Enabled) ] ,EQU(State,50) ]OTE(Error);
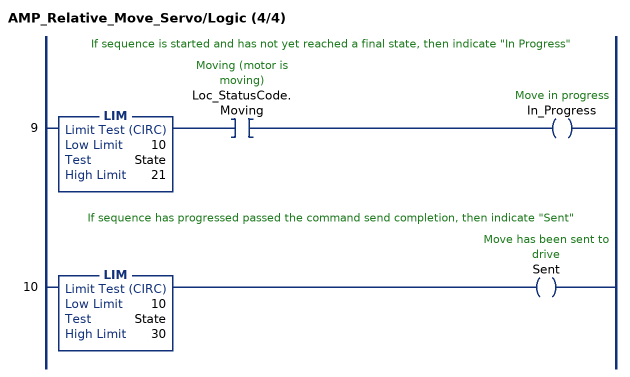
   // If sequence is started and has not yet reached a final state, then indicate "In Progress"
   9: LIM(10,State,21)XIC(Loc_StatusCode.Moving)OTE(In_Progress);
   // If sequence has progressed passed the command send completion, then indicate "Sent"
   10: LIM(10,State,30)OTE(Sent);
END_ROUTINE
END_ADD_ON_INSTRUCTION
